# EPICS IOC start-up script: examples/test/PSI/generic.iocsh
#- mXsXXX naming
require ecmccfg, "NAMING=mXsXXX"

#- add slaves
${SCRIPTEXEC} ${ecmccfg_DIR}addSlave.cmd, "HW_DESC=${HW}, SLAVE_ID=${SLAVE=0}"
